// TIA Portal V16 export
// export: Created 2023-07-30T20:35:41.3441687Z, ExportSetting WithDefaults, DisplayName Totally Integrated Automation Portal, DisplayVersion V16, DisplayName TIA Portal Version Control Interface, DisplayVersion V16, DisplayName TIA Portal Openness, DisplayVersion V16, DisplayName STEP 7 Professional, DisplayVersion V16, DisplayName STEP 7 Safety, DisplayVersion V16, DisplayName WinCC Professional, DisplayVersion V16
FUNCTION_BLOCK "modbuscomm"   // FB1, LAD
{ S7_Optimized_Access := 'TRUE' }
VERSION : 0.1
// stored: AutoNumber true, IsIECCheckEnabled false, IsRetainMemResEnabled false, MemoryReserve 100, SetENOAutomatically false, UDAEnableTagReadback false
   VAR_TEMP
      tag1 : Bool;
      tag2 : Bool;
   END_VAR
BEGIN

REGION Network 1
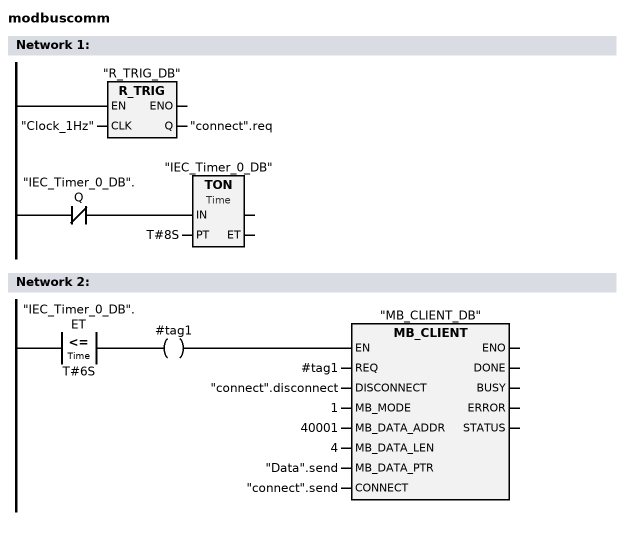
   RUNG wire#powerrail
      "R_TRIG_DB".R_TRIG(CLK := "Clock_1Hz", Q => "connect".req)
   END_RUNG
   RUNG wire#powerrail
      I_Contact( "IEC_Timer_0_DB".Q )
      { S7_Templates := "time_type := Time" } "IEC_Timer_0_DB".TON(pt := T#8S, et =>)
   END_RUNG
   // the same network as SCL:
   "R_TRIG_DB"(CLK := "Clock_1Hz", Q => "connect".req);   // R_TRIG
   "IEC_Timer_0_DB".TON(IN := NOT "IEC_Timer_0_DB".Q, PT := T#8S);
END_REGION

REGION Network 2
   RUNG wire#powerrail
      { S7_Templates := "SrcType := Time" } LE_Contact(in1 := "IEC_Timer_0_DB".ET, in2 := T#6S)
      Coil( #tag1 )
      "MB_CLIENT_DB".MB_CLIENT(REQ := #tag1, DISCONNECT := "connect".disconnect, MB_MODE := 1, MB_DATA_ADDR := 40001, MB_DATA_LEN := 4, MB_DATA_PTR := "Data".send, CONNECT := "connect".send, DONE =>, BUSY =>, ERROR =>, STATUS =>)
   END_RUNG
   // the same network as SCL:
   #tag1 := "IEC_Timer_0_DB".ET <= T#6S;
   IF #tag1 THEN
       "MB_CLIENT_DB"(REQ := #tag1,   // MB_CLIENT
                      DISCONNECT := "connect".disconnect,
                      MB_MODE := 1,
                      MB_DATA_ADDR := 40001,
                      MB_DATA_LEN := 4,
                      MB_DATA_PTR := "Data".send,
                      CONNECT := "connect".send);
   END_IF;
END_REGION
END_FUNCTION_BLOCK
